// TIA Portal V20 export
FUNCTION "{{BLOCK_NAME}}" : Void   // FC{{BLOCK_NUMBER}}, FBD
{ S7_Optimized_Access := 'TRUE' }
VERSION : 0.1
// stored: AutoNumber false, IsIECCheckEnabled false, SetENOAutomatically false
BEGIN

REGION Network 1: {{NETWORK_TITLE}}
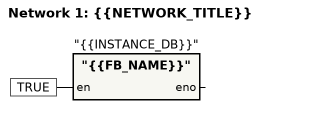
   IF TRUE THEN
       "{{INSTANCE_DB}}"();   // "{{FB_NAME}}"
   END_IF;
END_REGION
END_FUNCTION
